ADAPTER EVENT_HS_WSTRING (* Handshake pattern adapter interface with WSTRING payload: CNF/IND in, REQ/RSP out *)
  (* Standard: 61499-1; Description: Copyright (c) 2026 HR Agrartechnik GmbH This program and the accompanying materials are made available under the terms of the Eclipse Public License 2.0 which is available at https://www.eclipse.org/legal/epl-2.0/ SPDX-License-Identifier: EPL-2.0 *)
  (* Version 1.0, 2026-08-31, Franz Höpfinger, HR Agrartechnik GmbH, Data-carrying variant of EVENT_HS, matching Vyatkin's own 'service' adapter (Module 6, slide 48): same REQ/CNF/IND/RSP events, plus a WSTRING payload per event, exactly like the 'push,100' style messages in the slide's message-sequence examples (slide 42) *)
  PACKAGE adapter::types::bidirectional::Handshake;
  (* Documentation:
  Data-carrying variant of the Handshake design pattern adapter (IEC 61499 primer course, Module 6 – Design methods and patterns, Valeriy Vyatkin). Same REQ/CNF/IND/RSP event vocabulary as EVENT_HS, but each event carries a WSTRING payload – matching Vyatkin's own generic "service" adapter (slide 48), used throughout the Service-Oriented-Architecture part of the course for both service-requester and plant/process-data interfaces.
    - REQ / REQD – request + payload, from Plug to Socket (e.g. "push,100")
   - CNF / CNFD – confirmation + payload, from Socket to Plug, answers a REQ
   - IND / INDD – unsolicited indication + payload, from Socket to Plug
   - RSP / RSPD – response + payload, from Plug to Socket, answers an IND
    Same Socket/Plug role split as EVENT_HS: Plug (Name>>) plays the Requester/client role (fires REQ/RSP, reacts to CNF/IND); Socket (>>Name) plays the Responder/server role (reacts to REQ/RSP, fires CNF/IND).
   See test_AX/Meins/DesingPatterns/HandshakePattern/HandshakePattern.md for the full write-up; use this variant instead of the dataless EVENT_HS when an actual payload needs to travel with the handshake. The payload type is fixed at WSTRING for now and can be swapped for a more specific/typed adapter later if needed.
  *)
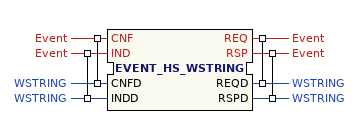
  EVENT_INPUT
    CNF WITH CNFD; (* Confirmation from Socket to Plug, answers a REQ *)
    IND WITH INDD; (* Indication from Socket to Plug *)
  END_EVENT
  EVENT_OUTPUT
    REQ WITH REQD; (* Request from Plug to Socket *)
    RSP WITH RSPD; (* Response from Plug to Socket, answers an IND *)
  END_EVENT
  VAR_INPUT
    CNFD : WSTRING; (* Confirmation payload, accompanies CNF *)
    INDD : WSTRING; (* Indication payload, accompanies IND *)
  END_VAR
  VAR_OUTPUT
    REQD : WSTRING; (* Request payload, accompanies REQ *)
    RSPD : WSTRING; (* Response payload, accompanies RSP *)
  END_VAR
  SERVICE PLUG/SOCKET
    SEQUENCE request_confirm
      PLUG.REQ(REQD) -> SOCKET.REQ(REQD);
      SOCKET.CNF(CNFD) -> PLUG.CNF(CNFD);
    END_SEQUENCE
    SEQUENCE indication_response
      SOCKET.IND(INDD) -> PLUG.IND(INDD);
      PLUG.RSP(RSPD) -> SOCKET.RSP(RSPD);
    END_SEQUENCE
  END_SERVICE
END_ADAPTER
